Omron CX-Programmer project NewProject (CX-Programmer 9.61)

# PLC NewPLC1: CP1E N30

## Global symbols (name address type ; comment)
0.00 BOOL  ; PB 1 START
0.01 BOOL  ; PB 2 STOP
100.00 BOOL  ; PILOT LAMP

## Program NewProgram1 (cyclic task 0)

### Section Section1

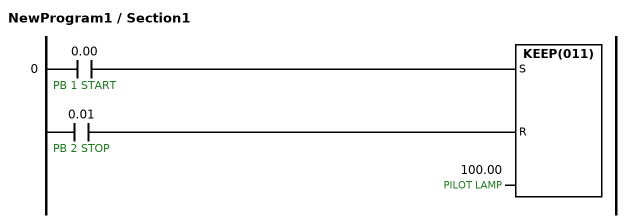
; rung 0
LD 0.00  ; PB 1 START
LD 0.01  ; PB 2 STOP
KEEP(011) 100.00  ; PILOT LAMP

### Section END
; rung 0
END(001)